// Mitsubishi GX Works2 project: 0702-1   PLC: Q02/Q02H

PROGRAM MAIN
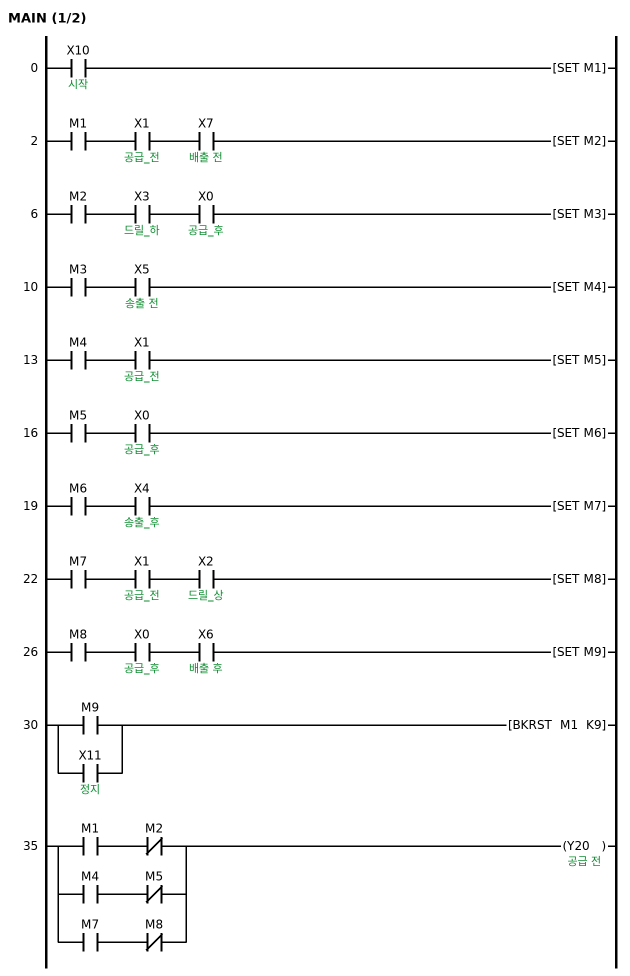
0     LD      X10  ; 시작
      SET     M1
2     LD      M1
      AND     X1  ; 공급_전
      AND     X7  ; 배출 전
      SET     M2
6     LD      M2
      AND     X3  ; 드릴_하
      AND     X0  ; 공급_후
      SET     M3
10    LD      M3
      AND     X5  ; 송출 전
      SET     M4
13    LD      M4
      AND     X1  ; 공급_전
      SET     M5
16    LD      M5
      AND     X0  ; 공급_후
      SET     M6
19    LD      M6
      AND     X4  ; 송출_후
      SET     M7
22    LD      M7
      AND     X1  ; 공급_전
      AND     X2  ; 드릴_상
      SET     M8
26    LD      M8
      AND     X0  ; 공급_후
      AND     X6  ; 배출 후
      SET     M9
30    LD      M9
      OR      X11  ; 정지
      BKRST   M1 K9
35    LD      M1
      ANI     M2
      LD      M4
      ANI     M5
      ORB
      LD      M7
      ANI     M8
      ORB
      OUT     Y20  ; 공급 전
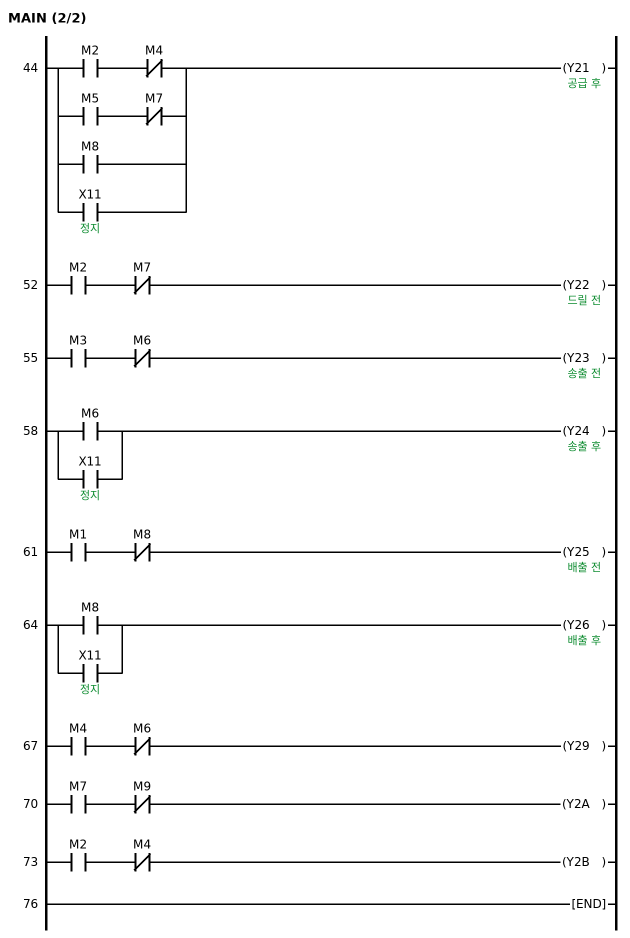
44    LD      M2
      ANI     M4
      LD      M5
      ANI     M7
      ORB
      OR      M8
      OR      X11  ; 정지
      OUT     Y21  ; 공급 후
52    LD      M2
      ANI     M7
      OUT     Y22  ; 드릴 전
55    LD      M3
      ANI     M6
      OUT     Y23  ; 송출 전
58    LD      M6
      OR      X11  ; 정지
      OUT     Y24  ; 송출 후
61    LD      M1
      ANI     M8
      OUT     Y25  ; 배출 전
64    LD      M8
      OR      X11  ; 정지
      OUT     Y26  ; 배출 후
67    LD      M4
      ANI     M6
      OUT     Y29
70    LD      M7
      ANI     M9
      OUT     Y2A
73    LD      M2
      ANI     M4
      OUT     Y2B
76    END
END_PROGRAM
